FUNCTION_BLOCK ConfigurationManager
  (* Standard: 61499-2 *)
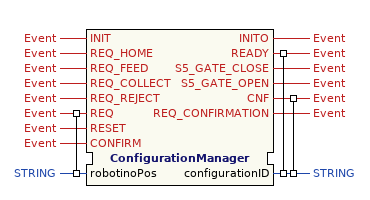
  EVENT_INPUT
    INIT;
    REQ_HOME;
    REQ_FEED;
    REQ_COLLECT;
    REQ_REJECT;
    REQ WITH robotinoPos;
    RESET;
    CONFIRM;
  END_EVENT
  EVENT_OUTPUT
    INITO;
    READY WITH configurationID;
    S5_GATE_CLOSE;
    S5_GATE_OPEN;
    CNF WITH configurationID;
    REQ_CONFIRMATION;
  END_EVENT
  VAR_INPUT
    robotinoPos : STRING;
  END_VAR
  VAR_OUTPUT
    configurationID : STRING;
  END_VAR
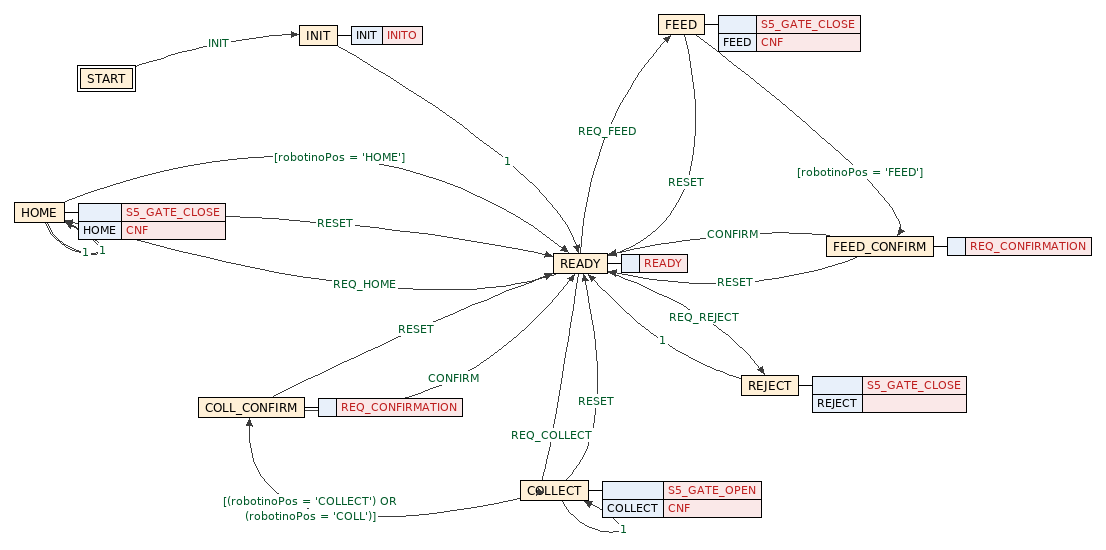
  EC_STATES
    START;
    INIT : INIT -> INITO;
    HOME : -> S5_GATE_CLOSE, HOME -> CNF;
    FEED : -> S5_GATE_CLOSE, FEED -> CNF;
    COLLECT : -> S5_GATE_OPEN, COLLECT -> CNF;
    REJECT : -> S5_GATE_CLOSE, REJECT;
    READY : -> READY;
    COLL_CONFIRM : -> REQ_CONFIRMATION;
    FEED_CONFIRM : -> REQ_CONFIRMATION;
  END_STATES
  EC_TRANSITIONS
    START TO INIT := INIT;
    INIT TO READY := 1;
    HOME TO READY := [robotinoPos = 'HOME'];
    READY TO HOME := REQ_HOME;
    READY TO COLLECT := REQ_COLLECT;
    COLLECT TO COLL_CONFIRM := [(robotinoPos = 'COLLECT') OR (robotinoPos = 'COLL')];
    READY TO REJECT := REQ_REJECT;
    REJECT TO READY := 1;
    READY TO FEED := REQ_FEED;
    FEED TO FEED_CONFIRM := [robotinoPos = 'FEED'];
    COLLECT TO READY := RESET;
    FEED TO READY := RESET;
    HOME TO READY := RESET;
    COLL_CONFIRM TO READY := CONFIRM;
    COLL_CONFIRM TO READY := RESET;
    FEED_CONFIRM TO READY := CONFIRM;
    FEED_CONFIRM TO READY := RESET;
    HOME TO HOME := 1;
    HOME TO HOME := 1;
    COLLECT TO COLLECT := 1;
  END_TRANSITIONS
  ALGORITHM INIT IN ST:
configurationID := 'NONE';&#10;
  END_ALGORITHM
  ALGORITHM HOME IN ST:
configurationID := 'HOME';&#10;
  END_ALGORITHM
  ALGORITHM FEED IN ST:
configurationID := 'FEED';&#10;
  END_ALGORITHM
  ALGORITHM COLLECT IN ST:
configurationID := 'COLLECT';&#10;
  END_ALGORITHM
  ALGORITHM REJECT IN ST:
configurationID := 'REJECT';&#10;
  END_ALGORITHM
END_FUNCTION_BLOCK
